FUNCTION_BLOCK ObserveCrane EXTENDS HardwareObservationBase
VAR_INPUT
END_VAR
VAR_OUTPUT
END_VAR
VAR
	m_ptrCrane: POINTER TO Crane;
	m_ptrCraneWP: POINTER TO xPPUProduct;
	
	m_rtAtStack: R_TRIG;
	m_rtAtLSC: R_TRIG;
	m_rtAtStamp: R_TRIG;
	
	m_resetCranePos: BOOL;
	
	// needed for a regression for the analog AngleDeg
	poti0: REAL;
	poti90: REAL;
	poti180: REAL;
END_VAR

METHOD FB_init : BOOL
VAR_INPUT
	bInitRetains : BOOL; // if TRUE, the retain variables are initialized (warm start / cold start)
	bInCopyCode : BOOL;  // if TRUE, the instance afterwards gets moved into the copy code (online change)

	i_ptrCrane: POINTER TO Crane;
	i_ptrWP: POINTER TO xPPUProduct;
END_VAR
m_ptrCrane := i_ptrCrane;
m_ptrCraneWP := i_ptrWP;
END_METHOD

METHOD  ResetDefinition : BOOL
VAR_INPUT
END_VAR
m_resetCranePos := TRUE;
END_METHOD

(* Update an instance of ProcessState with the part of the process that can be observed by this Hardware Interface. *)
METHOD UpdateProcessObservation : BOOL
VAR_IN_OUT
	io_processState: ProcessState;
END_VAR
VAR
	potiVal: REAL;
	x_bar: REAL;
	y_bar: REAL;
	a: REAL := -88.16748;		// initial value (calibrated 30 April 2025)
	b: REAL := 0.0129453959;	// initial value (calibrated 30 April 2025)
END_VAR
io_processState.UpdateState_Binary(EProcessVariables.Crane_AtStack, m_ptrCrane^.AtStack, i_force := TRUE);
io_processState.UpdateState_Binary(EProcessVariables.Crane_AtStamp, m_ptrCrane^.AtStamp, i_force := TRUE);
io_processState.UpdateState_Binary(EProcessVariables.Crane_AtLSC, m_ptrCrane^.AtConveyor, i_force := TRUE);
io_processState.UpdateState_Binary(EProcessVariables.Crane_HoldingWorkpiece, m_ptrCrane^.o_VacuumGripper.WPTaken, i_force := TRUE);
io_processState.UpdateState_Binary(EProcessVariables.Crane_CylinderExtended, m_ptrCrane^.o_MonostableCylinder.Extended, i_force := TRUE);
io_processState.UpdateState_Binary(EProcessVariables.Crane_CylinderRetracted, m_ptrCrane^.o_MonostableCylinder.Retracted, i_force := TRUE);

// Angle [in degrees] regression
potiVal := m_ptrCrane^.Motor.AI_Position;
IF m_ptrCrane^.AtStack THEN
	poti0 := potiVal;
ELSIF m_ptrCrane^.AtConveyor THEN
	poti90 := potiVal;
ELSIF m_ptrCrane^.AtStamp THEN
	poti180 := potiVal;
END_IF

IF poti0 <> 0 AND poti90 <> 0 AND poti180 <> 0 THEN
	x_bar := (poti0 + poti90 + poti180) / 3;
	y_bar := (90+180)/3;
	b := ((poti0 - x_bar)*-y_bar + (poti90 - x_bar)*(90 - y_bar) + (poti180 - x_bar)*(180 - y_bar))/
		(EXPT(poti0 - x_bar, 2) + EXPT(poti90 - x_bar, 2) + EXPT(poti180 - x_bar, 2));
	a := y_bar - b*x_bar;
ELSIF poti0 <> 0 AND poti90 <> 0 THEN
	x_bar := (poti0 + poti90) / 2;
	y_bar := 90/2;
	b := ((poti0 - x_bar)*-y_bar + (poti90 - x_bar)*(90 - y_bar))/
		(EXPT(poti0 - x_bar, 2) + EXPT(poti90 - x_bar, 2));
	a := y_bar - b*x_bar;
ELSIF poti90 <> 0 AND poti180 <> 0 THEN
	x_bar := (poti90 + poti180) / 2;
	y_bar := (90+180)/2;
	b := ((poti90 - x_bar)*(90 - y_bar) + (poti180 - x_bar)*(180 - y_bar))/
		(EXPT(poti90 - x_bar, 2) + EXPT(poti180 - x_bar, 2));
	a := y_bar - b*x_bar;
END_IF

io_processState.UpdateState_Numeric(EProcessVariables.Crane_Angle, a + b*potiVal, i_force := TRUE);

m_rtAtStack(CLK := m_ptrCrane^.AtStack);
m_rtAtStamp(CLK := m_ptrCrane^.AtStamp);
m_rtAtLSC(CLK := m_ptrCrane^.AtConveyor);

IF m_rtAtStack.Q OR m_rtAtStamp.Q OR m_rtAtLSC.Q THEN
	io_processState.UpdateState_Defined(EProcessVariables.Crane_AtStack, TRUE);
	io_processState.UpdateState_Defined(EProcessVariables.Crane_AtStamp, TRUE);
	io_processState.UpdateState_Defined(EProcessVariables.Crane_AtLSC, TRUE);
END_IF
IF m_resetCranePos THEN
	io_processState.UpdateState_Defined(EProcessVariables.Crane_AtStack, FALSE);
	io_processState.UpdateState_Defined(EProcessVariables.Crane_AtStamp, FALSE);
	io_processState.UpdateState_Defined(EProcessVariables.Crane_AtLSC, FALSE);
	m_resetCranePos := FALSE;
END_IF

io_processState.UpdateState_Defined(EProcessVariables.Crane_HoldingWorkpiece, TRUE);
io_processState.UpdateState_Defined(EProcessVariables.Crane_CylinderExtended, TRUE);
io_processState.UpdateState_Defined(EProcessVariables.Crane_CylinderRetracted, TRUE);
io_processState.UpdateState_Defined(EProcessVariables.Crane_Angle, TRUE);
END_METHOD

END_FUNCTION_BLOCK

(* stored: Version 1.1.0.1
   POU ObserveCrane: Id {787d945d-7a7b-490d-ac5b-e82218bdbe27}, SpecialFunc None
   Method FB_init: Id {dde86f07-4f6b-4aef-896a-b618b4ed962f}
   Method ResetDefinition: Id {81722e43-2499-410c-8b89-23dd0642fee1}
   Method UpdateProcessObservation: Id {eeabc617-6a60-4410-8f2d-ea0e6fac543c} *)
